TEXTLIST TextList_Type_Moteur
  0 = '' | FR: 'NU' | EN: 'NU'
  1 = '' | FR: 'Rotation PS' | EN: 'SH Rotation'
  2 = '' | FR: 'Translation PS' | EN: 'SH Translation'
  3 = '' | FR: 'Ascenseur' | EN: 'Stacker'
  4 = '' | FR: 'Rotation' | EN: 'Rotation'
  5 = '' | FR: 'Déploiement' | EN: 'Deployement'
  6 = '' | FR: 'Translation' | EN: 'Translation'
  7 = '' | FR: 'Porte Substrat' | EN: 'Substrate Holder'
  8 = '' | FR: 'Caches' | EN: 'Shutters'
  9 = '' | FR: 'Satellisation' | EN: 'Satellization'
  10 = '' | FR: 'Tilt Porte Substrat' | EN: 'Substrate holder Tilt'
   = ''
END_TEXTLIST

(* stored: Version 1.1.0.1, ProductVersion 3.1.4024.10
   TextList TextList_Type_Moteur: Id {29ed8b7c-ff4e-4461-bf44-fc9e20f05439} *)
